TYPE ST_Communication :
STRUCT
	
	ePackMLMode						: Tc3_PackML.E_PMLUnitMode;						//Mode 
	ePackMLAutoState				: Tc3_PackML.E_PMLState;							//PackML Auto State
	sPackMLCommand					: ST_PackMLCmdForCom;					//PackML Commands
	
	eError							: S_Error;
	
	bEnable							: BOOL;	
	bCycleStart						: BOOL;
	bCycleStop						: BOOL;
	bCycleReset						: BOOL;
	bManualMode						: BOOL;
	bHoming							: BOOL;
	bHomingDone						: BOOL;	
	bConfectionEnding				: BOOL;
	tCycleTime						: TIME;
	iWatchdog						: INT;
	
	sRecipeName						: STRING(255);							
	sRecipeIndex					: STRING(255);
	
	eMachinePermissions				: ST_MachinePermissions;
	eReservedSignals				: ST_ReservedSignals;
END_STRUCT
END_TYPE

(* stored: Version 1.1.0.1, ProductVersion 3.1.4026.13, FileIdentifier 0025bea97517f9f7be374d71b7a25751c56141ef, FileSignature 905d5696aa1623a516eff6b172c2a7d5913ab69dc6a2e9f49dba85c2b8f38c9d67cdf43cabd435137b2be8ac0d4a8b9968c1154c06df34b9b06817e0fb5e3a5fb5feae8d2280d93e8dfa56bb2c85aaab7a185d6be1487f3401650b64a12cc2ed0c73706668d1a5f8278ad6f5ad63ff80beef2fd2ee6b1910a556b4b95941eb05f7515acb5fada70e15b05a4c481aecc88c001dbabe064a466edcb6e8846f9e63e45bdd6b4eea381bf2088ed3566b578c2eac33f0ed0e5af7eaa971364817dd69b04630ef92cbccf136eb4df3260dc83da3c19c055ef536d5ac66a2ef6690d8257723abe18c27ba14984f5fc1622c95801158d2f402be7f05b43e56e64f599687
   DUT ST_Communication: Id {6513464b-4f6b-418b-a7a1-d62ac1164468} *)
